FUNCTION_BLOCK XtsFacade
VAR
	group : XtsCAGroup;
	hardware : XtsHardware;
	movers : ARRAY[0..10] OF XtsMover;
	stations : ARRAY[0..5] OF XtsStations;
	xpu : XtsXPU;
	i: INT;
	InitState : INT;
END_VAR

METHOD InitialiseXts : BOOL
VAR_INPUT
END_VAR
VAR
	InitCheck : BOOL;
END_VAR
CASE InitState OF
	0: 
		IF group.AddMoverToGroup() THEN
			InitState := 10;
		END_IF
	10:
		IF xpu.GetMoverInterface() THEN
			InitState := 20;
		END_IF
	20:
		InitCheck := TRUE;
		FOR i := 0 TO 5 DO
			InitCheck := InitCheck AND stations[i].InitialiseStation();
		END_FOR
		IF InitCheck THEN
			InitState := 30;
		END_IF
	30:
		IF hardware.CheckModuleVoltages() THEN
			InitState := 40;
		END_IF
	40:
		InitialiseXts := true;
END_CASE


hardware.CheckModuleVoltages();
END_METHOD

END_FUNCTION_BLOCK

(* stored: Version 1.1.0.1, ProductVersion 3.1.4024.12
   POU XtsFacade: Id {0fde9a4f-e82c-4e21-9129-4ed3d18c8355}, SpecialFunc None
   Method InitialiseXts: Id {d0208558-6e71-4e3f-aa75-da36fa295b0d} *)
